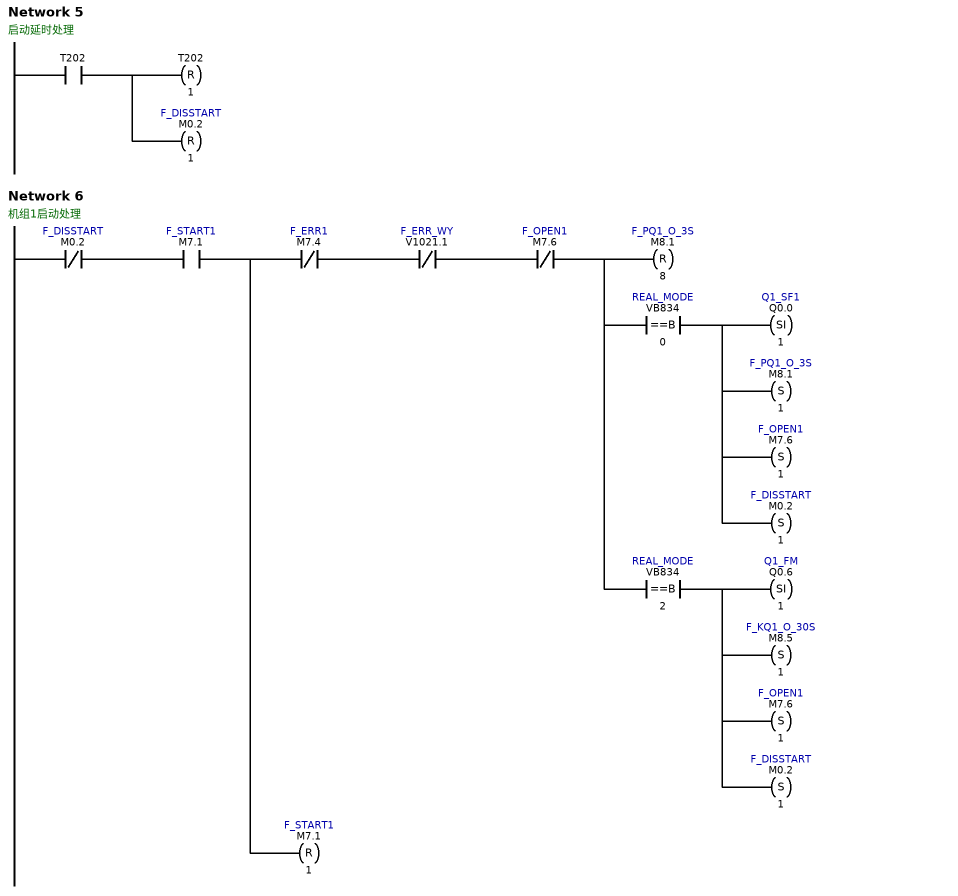
[picture p48: SBR7 networks 5-6]
Network 5
// 启动延时处理
LD     T202
R      T202, 1
R      F_DISSTART:M0.2, 1
Network 6
// 机组1启动处理
LDN    F_DISSTART:M0.2
A      F_START1:M7.1
LPS
AN     F_ERR1:M7.4
AN     F_ERR_WY:V1021.1
AN     F_OPEN1:M7.6
LPS
R      F_PQ1_O_3S:M8.1, 8
AB=    REAL_MODE:VB834, 0
SI     Q1_SF1:Q0.0, 1
S      F_PQ1_O_3S:M8.1, 1
S      F_OPEN1:M7.6, 1
S      F_DISSTART:M0.2, 1
LPP
AB=    REAL_MODE:VB834, 2
SI     Q1_FM:Q0.6, 1
S      F_KQ1_O_30S:M8.5, 1
S      F_OPEN1:M7.6, 1
S      F_DISSTART:M0.2, 1
LPP
R      F_START1:M7.1, 1
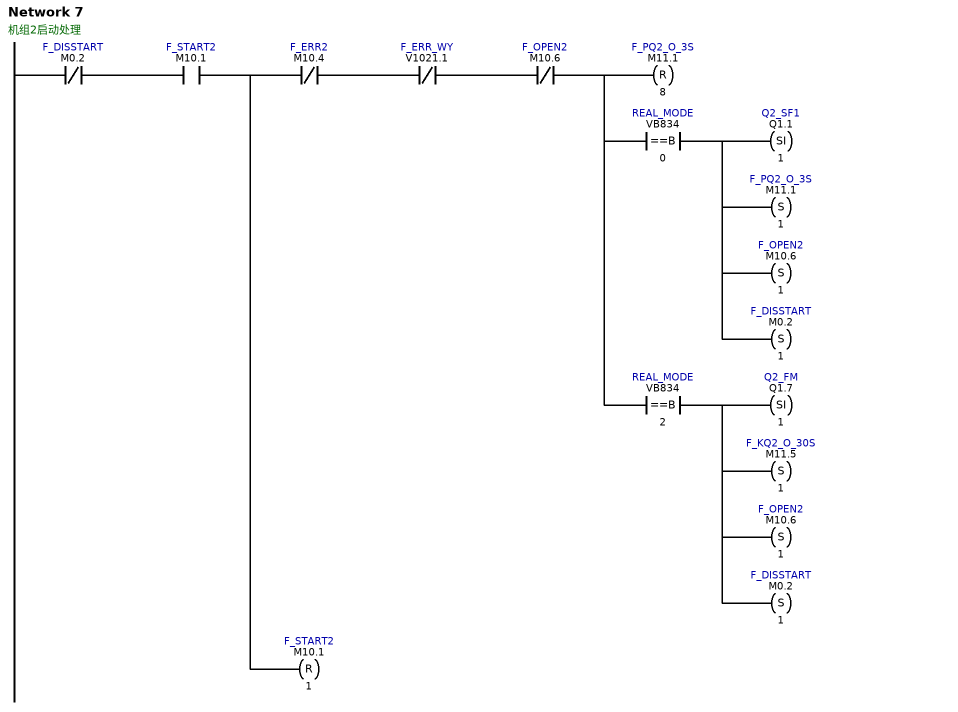
Network 7
// 机组2启动处理
LDN    F_DISSTART:M0.2
A      F_START2:M10.1
LPS
AN     F_ERR2:M10.4
AN     F_ERR_WY:V1021.1
AN     F_OPEN2:M10.6
LPS
R      F_PQ2_O_3S:M11.1, 8
AB=    REAL_MODE:VB834, 0
SI     Q2_SF1:Q1.1, 1
S      F_PQ2_O_3S:M11.1, 1
S      F_OPEN2:M10.6, 1
S      F_DISSTART:M0.2, 1
LPP
AB=    REAL_MODE:VB834, 2
SI     Q2_FM:Q1.7, 1
S      F_KQ2_O_30S:M11.5, 1
S      F_OPEN2:M10.6, 1
S      F_DISSTART:M0.2, 1
LPP
R      F_START2:M10.1, 1
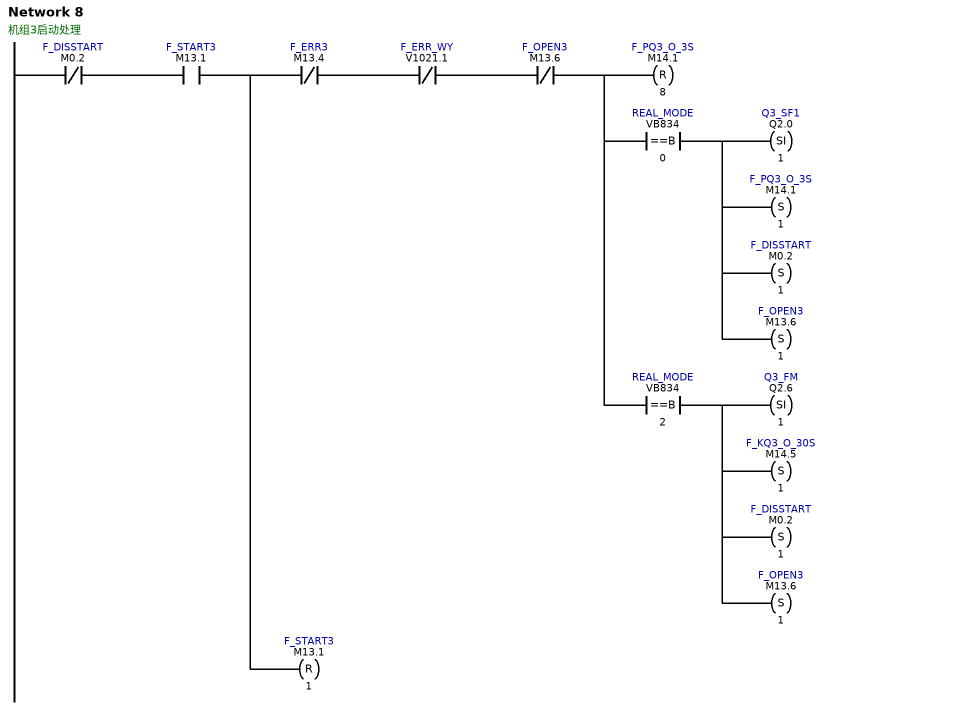
Network 8
// 机组3启动处理
LDN    F_DISSTART:M0.2
A      F_START3:M13.1
LPS
AN     F_ERR3:M13.4
AN     F_ERR_WY:V1021.1
AN     F_OPEN3:M13.6
LPS
R      F_PQ3_O_3S:M14.1, 8
AB=    REAL_MODE:VB834, 0
SI     Q3_SF1:Q2.0, 1
S      F_PQ3_O_3S:M14.1, 1
S      F_DISSTART:M0.2, 1
S      F_OPEN3:M13.6, 1
LPP
AB=    REAL_MODE:VB834, 2
SI     Q3_FM:Q2.6, 1
S      F_KQ3_O_30S:M14.5, 1
S      F_DISSTART:M0.2, 1
S      F_OPEN3:M13.6, 1
LPP
R      F_START3:M13.1, 1
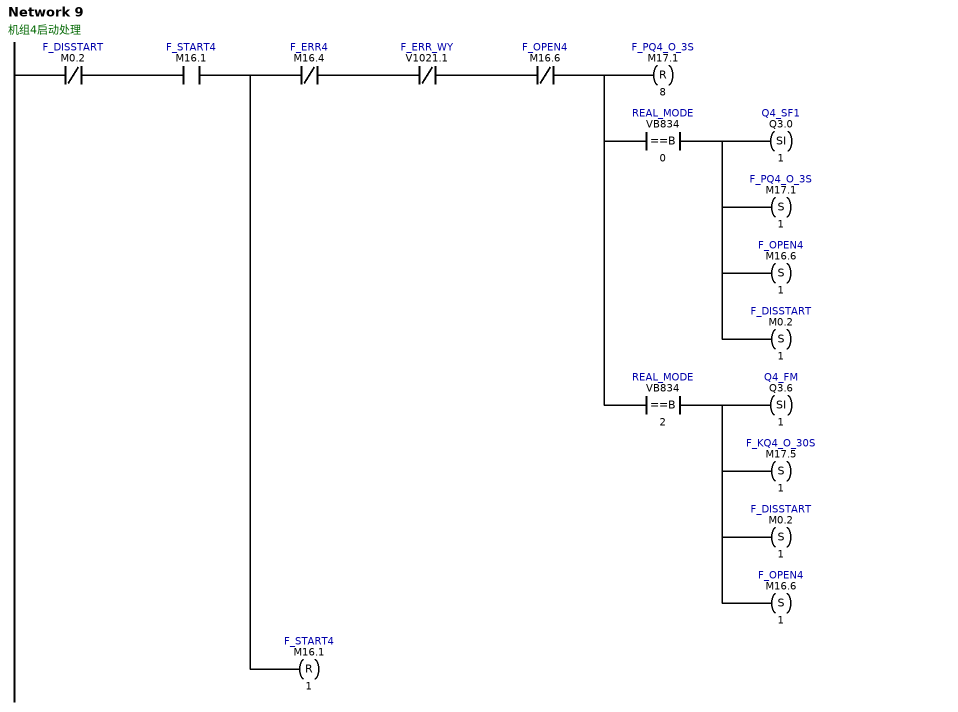
Network 9
// 机组4启动处理
LDN    F_DISSTART:M0.2
A      F_START4:M16.1
LPS
AN     F_ERR4:M16.4
AN     F_ERR_WY:V1021.1
AN     F_OPEN4:M16.6
LPS
R      F_PQ4_O_3S:M17.1, 8
AB=    REAL_MODE:VB834, 0
SI     Q4_SF1:Q3.0, 1
S      F_PQ4_O_3S:M17.1, 1
S      F_OPEN4:M16.6, 1
S      F_DISSTART:M0.2, 1
LPP
AB=    REAL_MODE:VB834, 2
SI     Q4_FM:Q3.6, 1
S      F_KQ4_O_30S:M17.5, 1
S      F_DISSTART:M0.2, 1
S      F_OPEN4:M16.6, 1
LPP
R      F_START4:M16.1, 1
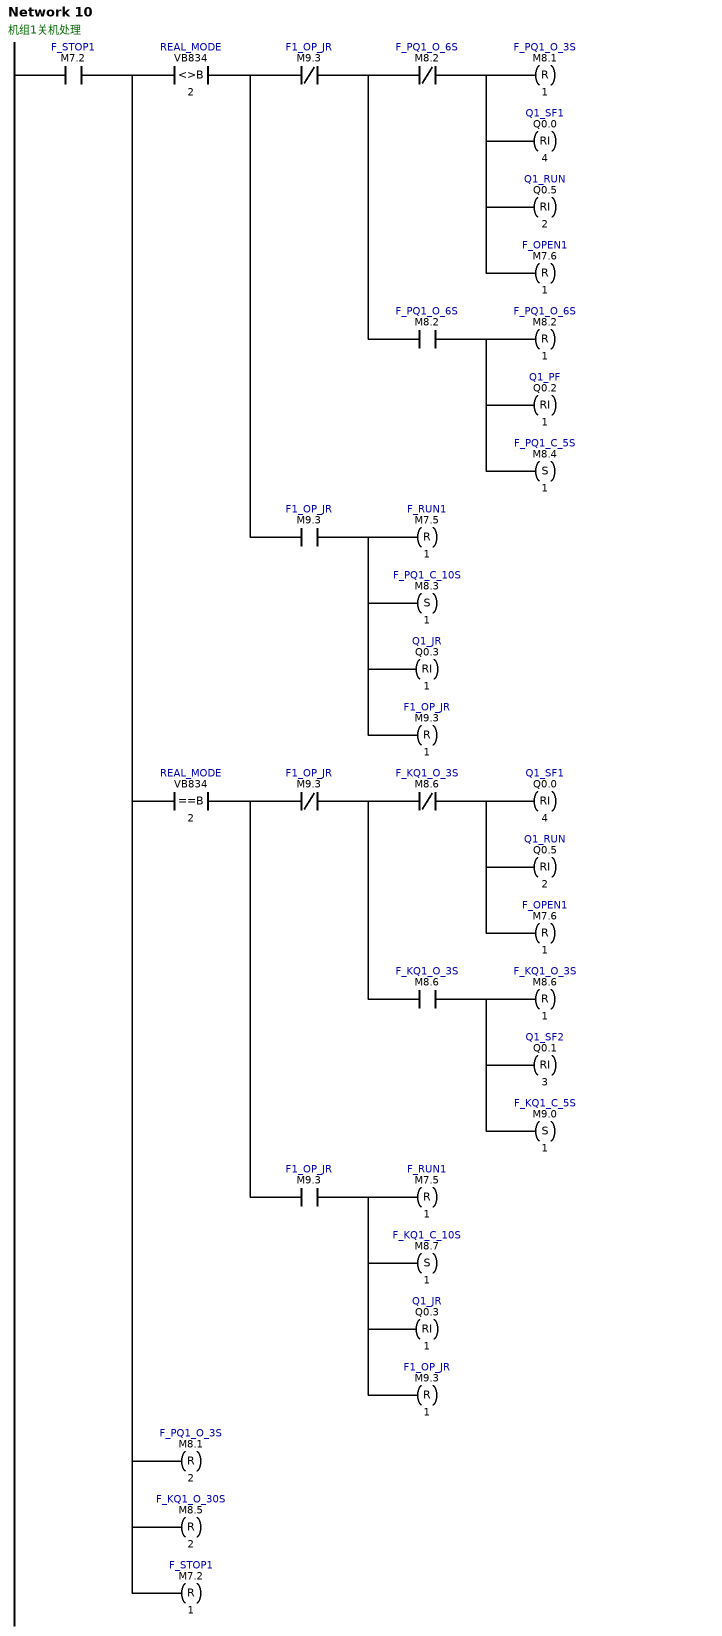
Network 10
// 机组1关机处理
LD     F_STOP1:M7.2
LPS
AB<>   REAL_MODE:VB834, 2
LPS
AN     F1_OP_JR:M9.3
LPS
AN     F_PQ1_O_6S:M8.2
R      F_PQ1_O_3S:M8.1, 1
RI     Q1_SF1:Q0.0, 4
RI     Q1_RUN:Q0.5, 2
R      F_OPEN1:M7.6, 1
LPP
A      F_PQ1_O_6S:M8.2
R      F_PQ1_O_6S:M8.2, 1
RI     Q1_PF:Q0.2, 1
S      F_PQ1_C_5S:M8.4, 1
LPP
A      F1_OP_JR:M9.3
R      F_RUN1:M7.5, 1
S      F_PQ1_C_10S:M8.3, 1
RI     Q1_JR:Q0.3, 1
R      F1_OP_JR:M9.3, 1
LRD
AB=    REAL_MODE:VB834, 2
LPS
AN     F1_OP_JR:M9.3
LPS
AN     F_KQ1_O_3S:M8.6
RI     Q1_SF1:Q0.0, 4
RI     Q1_RUN:Q0.5, 2
R      F_OPEN1:M7.6, 1
LPP
A      F_KQ1_O_3S:M8.6
R      F_KQ1_O_3S:M8.6, 1
RI     Q1_SF2:Q0.1, 3
S      F_KQ1_C_5S:M9.0, 1
LPP
A      F1_OP_JR:M9.3
R      F_RUN1:M7.5, 1
S      F_KQ1_C_10S:M8.7, 1
RI     Q1_JR:Q0.3, 1
R      F1_OP_JR:M9.3, 1
LPP
R      F_PQ1_O_3S:M8.1, 2
R      F_KQ1_O_30S:M8.5, 2
R      F_STOP1:M7.2, 1
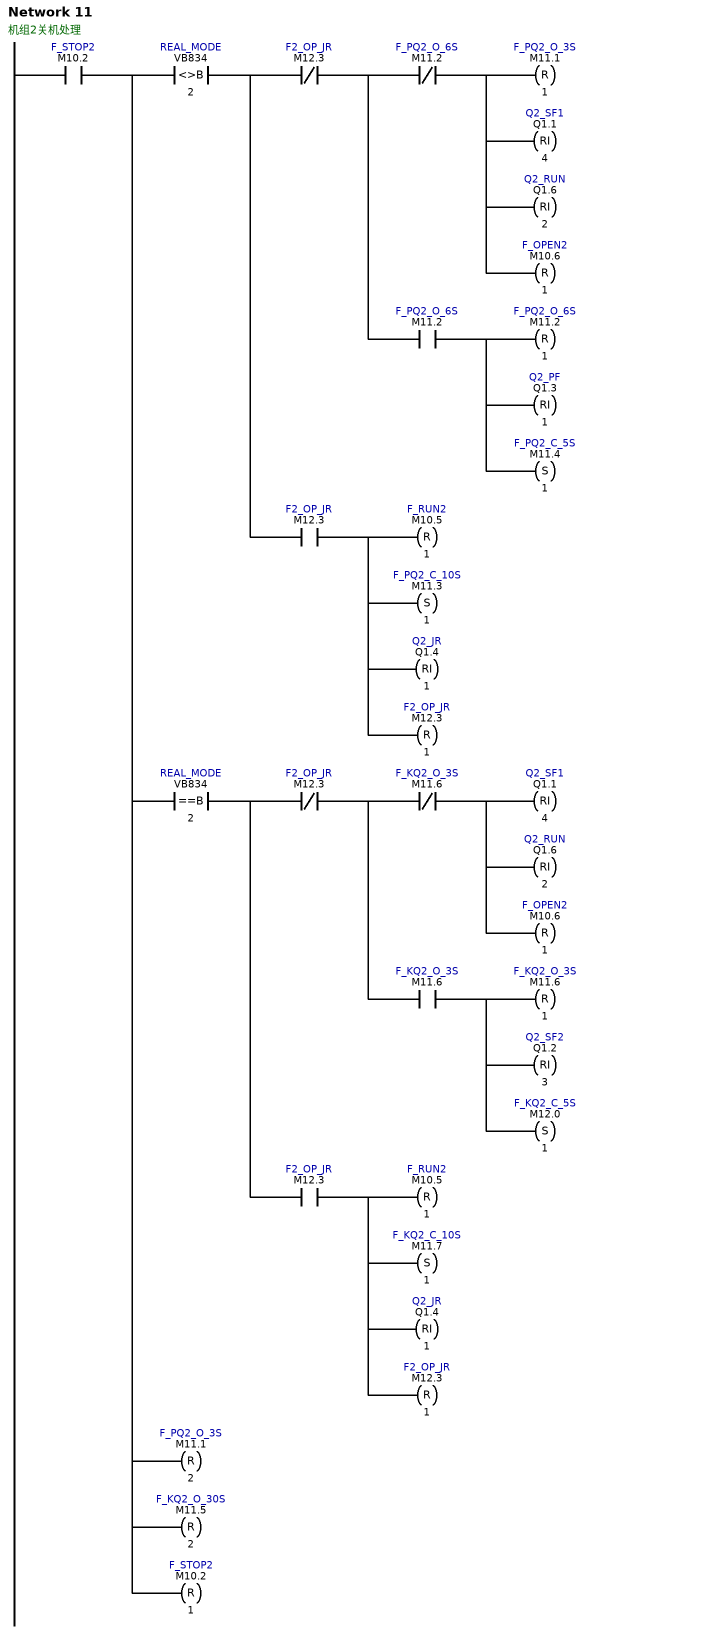
Network 11
// 机组2关机处理
LD     F_STOP2:M10.2
LPS
AB<>   REAL_MODE:VB834, 2
LPS
AN     F2_OP_JR:M12.3
LPS
AN     F_PQ2_O_6S:M11.2
R      F_PQ2_O_3S:M11.1, 1
RI     Q2_SF1:Q1.1, 4
RI     Q2_RUN:Q1.6, 2
R      F_OPEN2:M10.6, 1
LPP
A      F_PQ2_O_6S:M11.2
R      F_PQ2_O_6S:M11.2, 1
RI     Q2_PF:Q1.3, 1
S      F_PQ2_C_5S:M11.4, 1
LPP
A      F2_OP_JR:M12.3
R      F_RUN2:M10.5, 1
S      F_PQ2_C_10S:M11.3, 1
RI     Q2_JR:Q1.4, 1
R      F2_OP_JR:M12.3, 1
LRD
AB=    REAL_MODE:VB834, 2
LPS
AN     F2_OP_JR:M12.3
LPS
AN     F_KQ2_O_3S:M11.6
RI     Q2_SF1:Q1.1, 4
RI     Q2_RUN:Q1.6, 2
R      F_OPEN2:M10.6, 1
LPP
A      F_KQ2_O_3S:M11.6
R      F_KQ2_O_3S:M11.6, 1
RI     Q2_SF2:Q1.2, 3
S      F_KQ2_C_5S:M12.0, 1
LPP
A      F2_OP_JR:M12.3
R      F_RUN2:M10.5, 1
S      F_KQ2_C_10S:M11.7, 1
RI     Q2_JR:Q1.4, 1
R      F2_OP_JR:M12.3, 1
LPP
R      F_PQ2_O_3S:M11.1, 2
R      F_KQ2_O_30S:M11.5, 2
R      F_STOP2:M10.2, 1
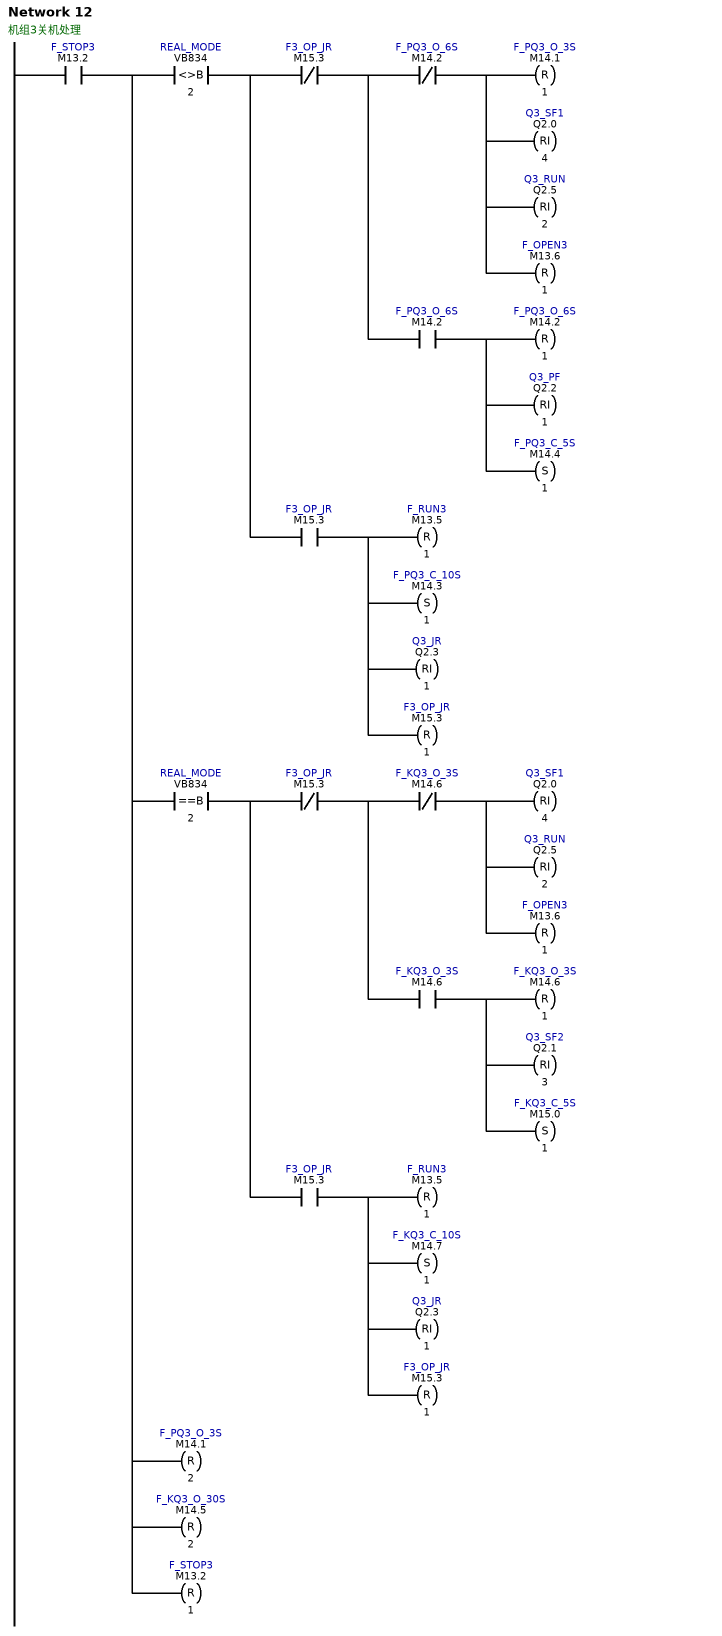
Network 12
// 机组3关机处理
LD     F_STOP3:M13.2
LPS
AB<>   REAL_MODE:VB834, 2
LPS
AN     F3_OP_JR:M15.3
LPS
AN     F_PQ3_O_6S:M14.2
R      F_PQ3_O_3S:M14.1, 1
RI     Q3_SF1:Q2.0, 4
RI     Q3_RUN:Q2.5, 2
R      F_OPEN3:M13.6, 1
LPP
A      F_PQ3_O_6S:M14.2
R      F_PQ3_O_6S:M14.2, 1
RI     Q3_PF:Q2.2, 1
S      F_PQ3_C_5S:M14.4, 1
LPP
A      F3_OP_JR:M15.3
R      F_RUN3:M13.5, 1
S      F_PQ3_C_10S:M14.3, 1
RI     Q3_JR:Q2.3, 1
R      F3_OP_JR:M15.3, 1
LRD
AB=    REAL_MODE:VB834, 2
LPS
AN     F3_OP_JR:M15.3
LPS
AN     F_KQ3_O_3S:M14.6
RI     Q3_SF1:Q2.0, 4
RI     Q3_RUN:Q2.5, 2
R      F_OPEN3:M13.6, 1
LPP
A      F_KQ3_O_3S:M14.6
R      F_KQ3_O_3S:M14.6, 1
RI     Q3_SF2:Q2.1, 3
S      F_KQ3_C_5S:M15.0, 1
LPP
A      F3_OP_JR:M15.3
R      F_RUN3:M13.5, 1
S      F_KQ3_C_10S:M14.7, 1
RI     Q3_JR:Q2.3, 1
R      F3_OP_JR:M15.3, 1
LPP
R      F_PQ3_O_3S:M14.1, 2
R      F_KQ3_O_30S:M14.5, 2
R      F_STOP3:M13.2, 1
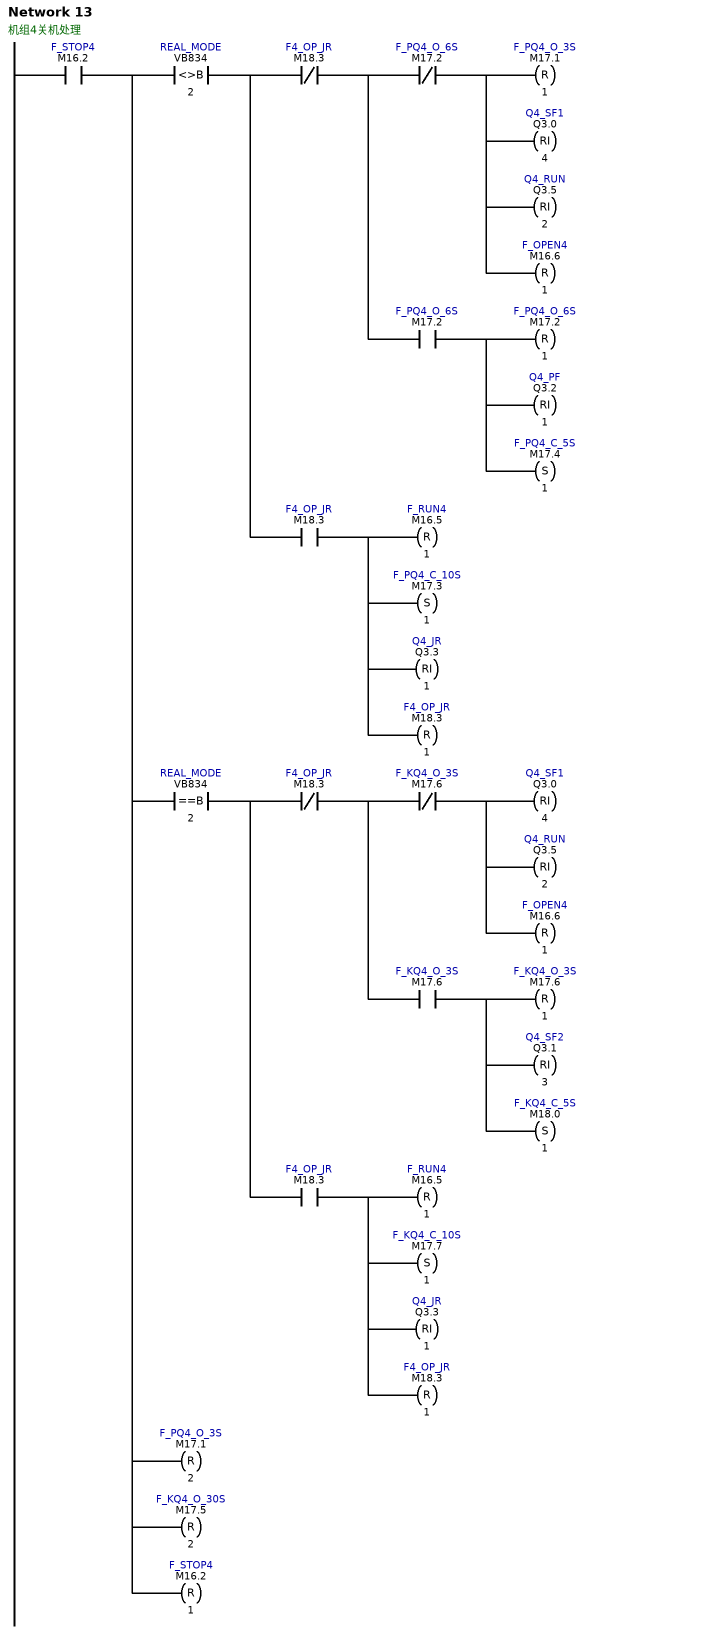
Network 13
// 机组4关机处理
LD     F_STOP4:M16.2
LPS
AB<>   REAL_MODE:VB834, 2
LPS
AN     F4_OP_JR:M18.3
LPS
AN     F_PQ4_O_6S:M17.2
R      F_PQ4_O_3S:M17.1, 1
RI     Q4_SF1:Q3.0, 4
RI     Q4_RUN:Q3.5, 2
R      F_OPEN4:M16.6, 1
LPP
A      F_PQ4_O_6S:M17.2
R      F_PQ4_O_6S:M17.2, 1
RI     Q4_PF:Q3.2, 1
S      F_PQ4_C_5S:M17.4, 1
LPP
A      F4_OP_JR:M18.3
R      F_RUN4:M16.5, 1
S      F_PQ4_C_10S:M17.3, 1
RI     Q4_JR:Q3.3, 1
R      F4_OP_JR:M18.3, 1
LRD
AB=    REAL_MODE:VB834, 2
LPS
AN     F4_OP_JR:M18.3
LPS
AN     F_KQ4_O_3S:M17.6
RI     Q4_SF1:Q3.0, 4
RI     Q4_RUN:Q3.5, 2
R      F_OPEN4:M16.6, 1
LPP
A      F_KQ4_O_3S:M17.6
R      F_KQ4_O_3S:M17.6, 1
RI     Q4_SF2:Q3.1, 3
S      F_KQ4_C_5S:M18.0, 1
LPP
A      F4_OP_JR:M18.3
R      F_RUN4:M16.5, 1
S      F_KQ4_C_10S:M17.7, 1
RI     Q4_JR:Q3.3, 1
R      F4_OP_JR:M18.3, 1
LPP
R      F_PQ4_O_3S:M17.1, 2
R      F_KQ4_O_30S:M17.5, 2
R      F_STOP4:M16.2, 1
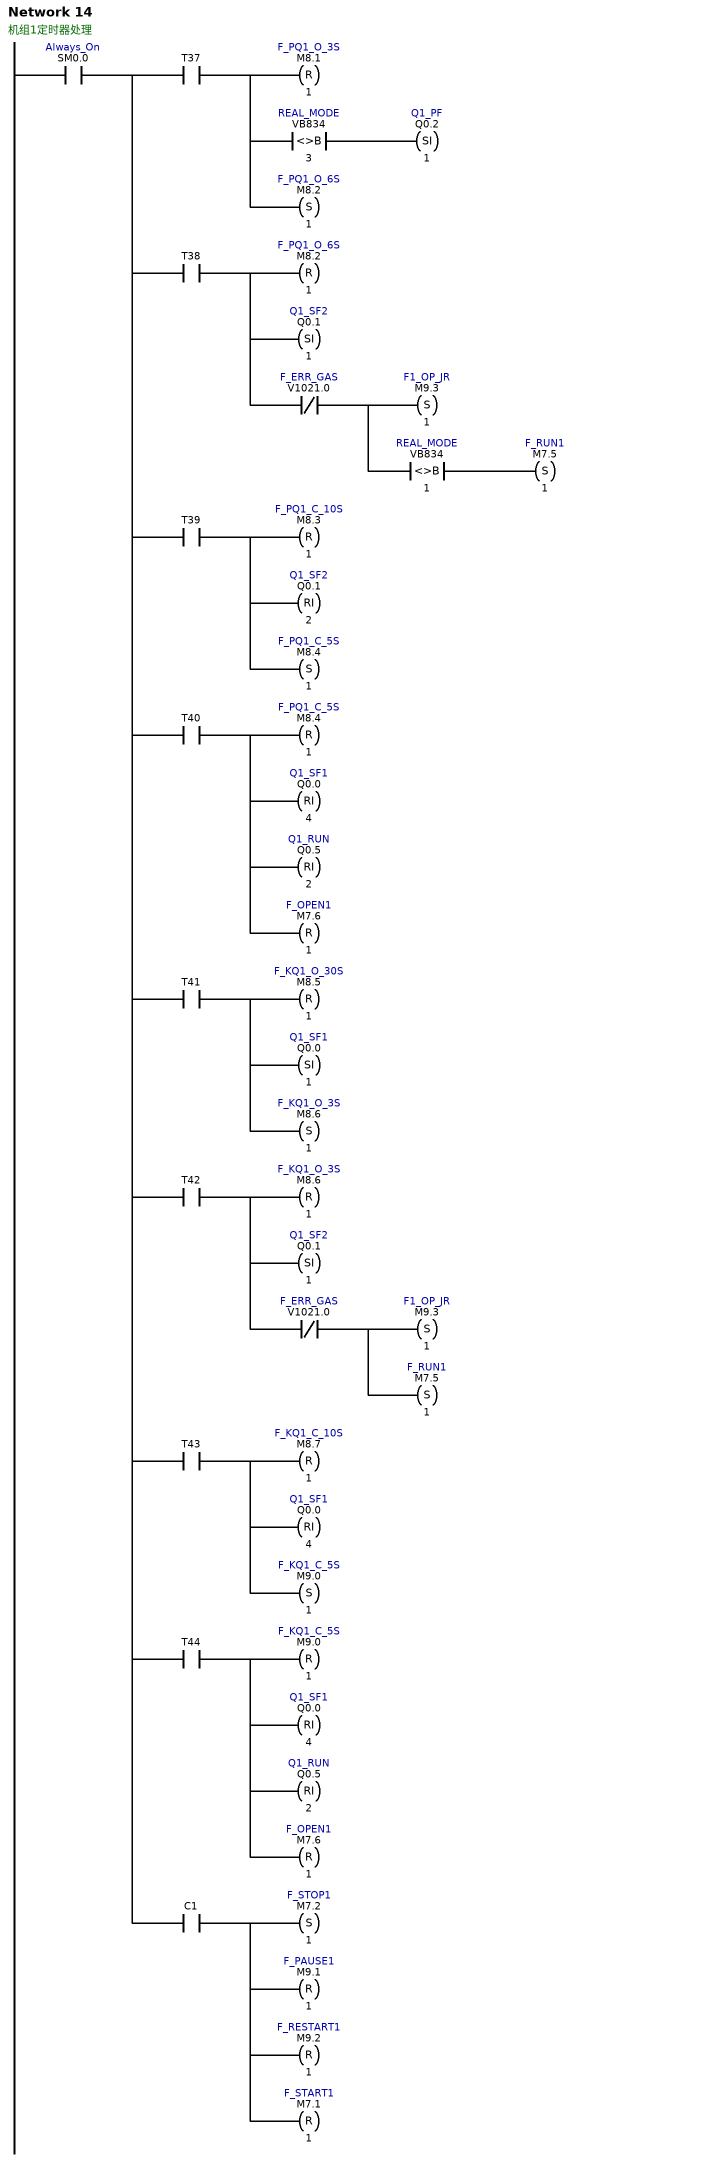
Network 14
// 机组1定时器处理
LD     Always_On:SM0.0
LPS
A      T37
LPS
R      F_PQ1_O_3S:M8.1, 1
AB<>   REAL_MODE:VB834, 3
SI     Q1_PF:Q0.2, 1
LPP
S      F_PQ1_O_6S:M8.2, 1
LRD
A      T38
R      F_PQ1_O_6S:M8.2, 1
SI     Q1_SF2:Q0.1, 1
AN     F_ERR_GAS:V1021.0
S      F1_OP_JR:M9.3, 1
AB<>   REAL_MODE:VB834, 1
S      F_RUN1:M7.5, 1
LRD
LPS
A      T39
R      F_PQ1_C_10S:M8.3, 1
RI     Q1_SF2:Q0.1, 2
S      F_PQ1_C_5S:M8.4, 1
LRD
A      T40
R      F_PQ1_C_5S:M8.4, 1
RI     Q1_SF1:Q0.0, 4
RI     Q1_RUN:Q0.5, 2
R      F_OPEN1:M7.6, 1
LPP
A      T41
R      F_KQ1_O_30S:M8.5, 1
SI     Q1_SF1:Q0.0, 1
S      F_KQ1_O_3S:M8.6, 1
LRD
A      T42
R      F_KQ1_O_3S:M8.6, 1
SI     Q1_SF2:Q0.1, 1
AN     F_ERR_GAS:V1021.0
S      F1_OP_JR:M9.3, 1
S      F_RUN1:M7.5, 1
LPP
LPS
A      T43
R      F_KQ1_C_10S:M8.7, 1
RI     Q1_SF1:Q0.0, 4
S      F_KQ1_C_5S:M9.0, 1
LRD
A      T44
R      F_KQ1_C_5S:M9.0, 1
RI     Q1_SF1:Q0.0, 4
RI     Q1_RUN:Q0.5, 2
R      F_OPEN1:M7.6, 1
LPP
A      C1
S      F_STOP1:M7.2, 1
R      F_PAUSE1:M9.1, 1
R      F_RESTART1:M9.2, 1
R      F_START1:M7.1, 1
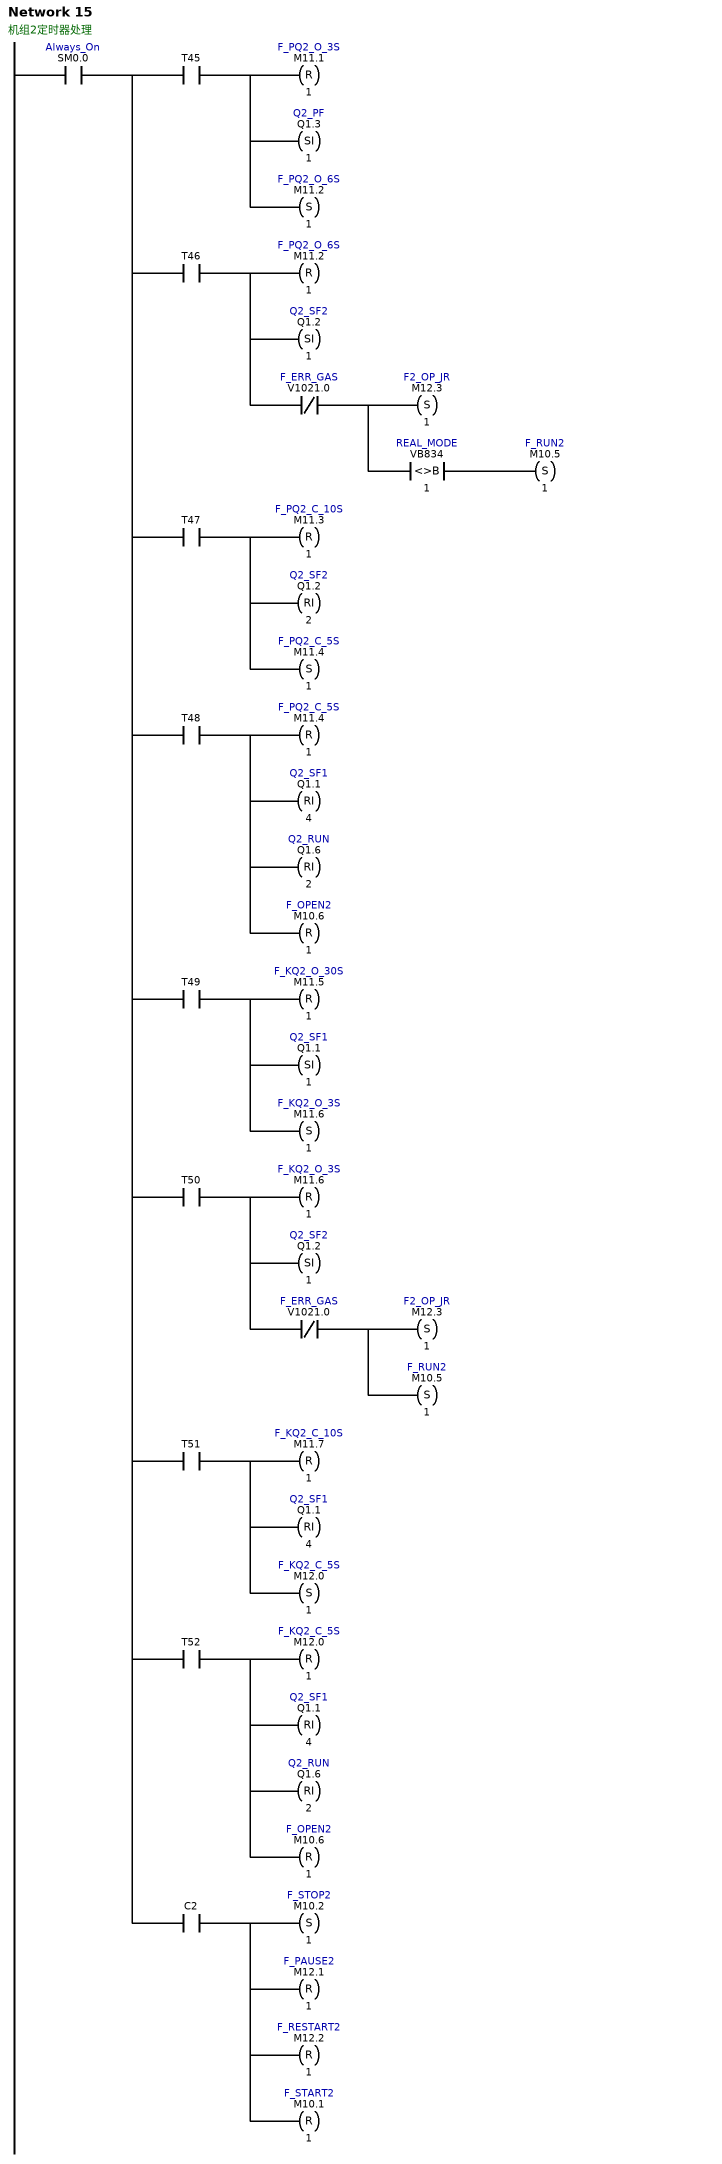
Network 15
// 机组2定时器处理
LD     Always_On:SM0.0
LPS
A      T45
R      F_PQ2_O_3S:M11.1, 1
SI     Q2_PF:Q1.3, 1
S      F_PQ2_O_6S:M11.2, 1
LRD
A      T46
R      F_PQ2_O_6S:M11.2, 1
SI     Q2_SF2:Q1.2, 1
AN     F_ERR_GAS:V1021.0
S      F2_OP_JR:M12.3, 1
AB<>   REAL_MODE:VB834, 1
S      F_RUN2:M10.5, 1
LRD
LPS
A      T47
R      F_PQ2_C_10S:M11.3, 1
RI     Q2_SF2:Q1.2, 2
S      F_PQ2_C_5S:M11.4, 1
LRD
A      T48
R      F_PQ2_C_5S:M11.4, 1
RI     Q2_SF1:Q1.1, 4
RI     Q2_RUN:Q1.6, 2
R      F_OPEN2:M10.6, 1
LPP
A      T49
R      F_KQ2_O_30S:M11.5, 1
SI     Q2_SF1:Q1.1, 1
S      F_KQ2_O_3S:M11.6, 1
LRD
A      T50
R      F_KQ2_O_3S:M11.6, 1
SI     Q2_SF2:Q1.2, 1
AN     F_ERR_GAS:V1021.0
S      F2_OP_JR:M12.3, 1
S      F_RUN2:M10.5, 1
LPP
LPS
A      T51
R      F_KQ2_C_10S:M11.7, 1
RI     Q2_SF1:Q1.1, 4
S      F_KQ2_C_5S:M12.0, 1
LRD
A      T52
R      F_KQ2_C_5S:M12.0, 1
RI     Q2_SF1:Q1.1, 4
RI     Q2_RUN:Q1.6, 2
R      F_OPEN2:M10.6, 1
LPP
A      C2
S      F_STOP2:M10.2, 1
R      F_PAUSE2:M12.1, 1
R      F_RESTART2:M12.2, 1
R      F_START2:M10.1, 1
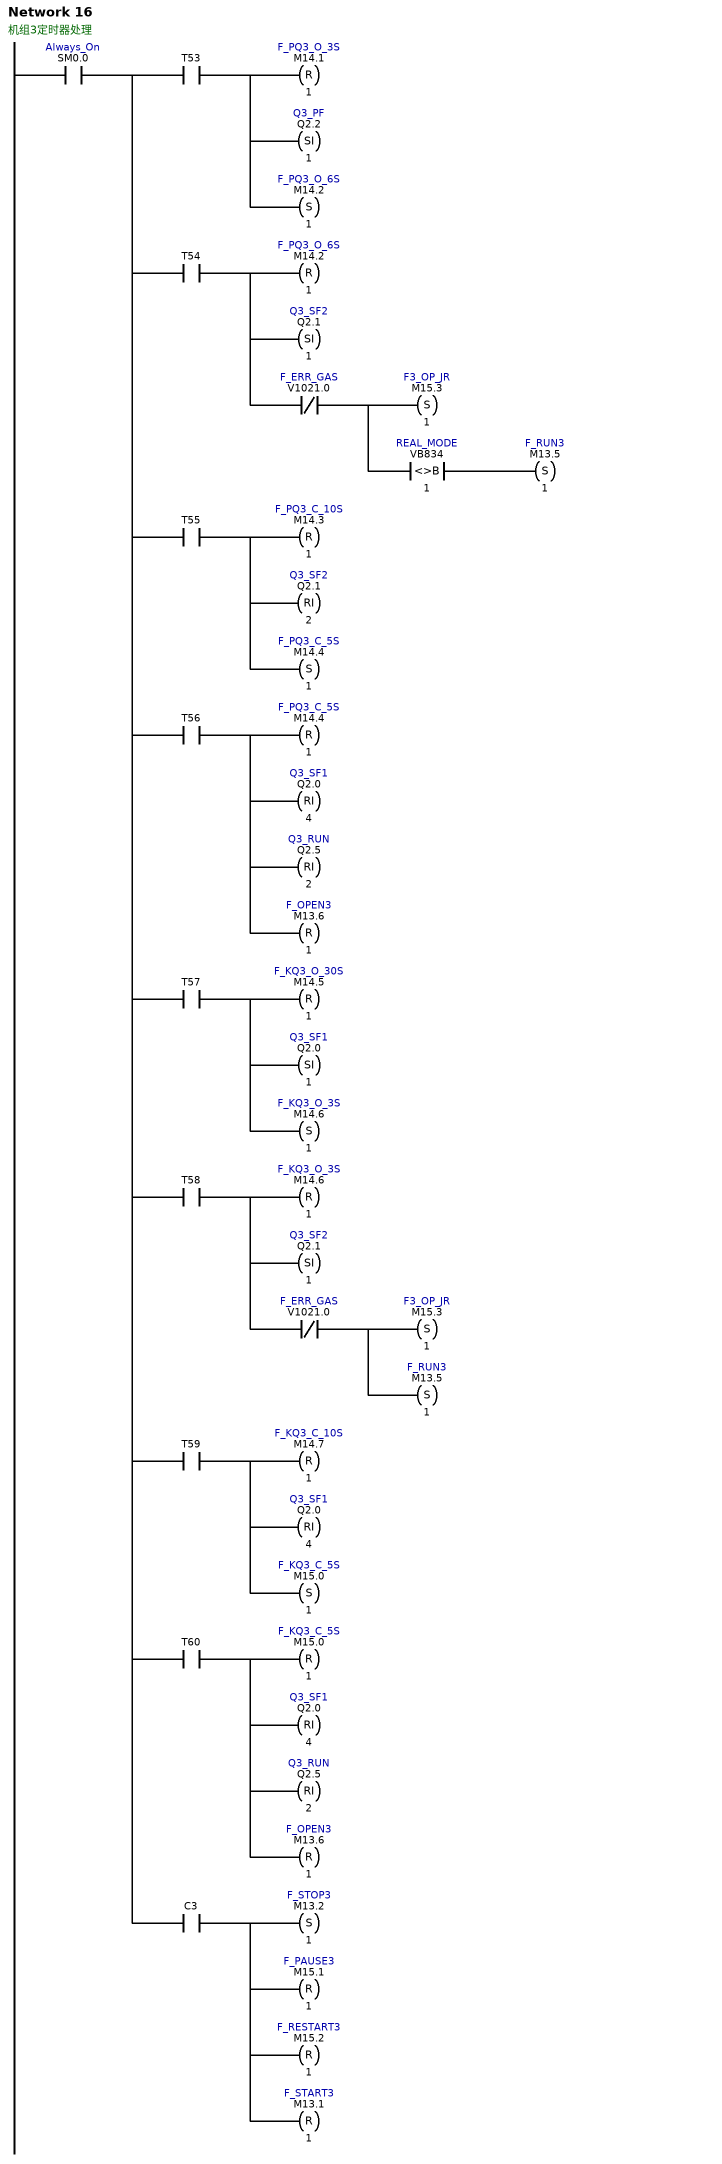
Network 16
// 机组3定时器处理
LD     Always_On:SM0.0
LPS
A      T53
R      F_PQ3_O_3S:M14.1, 1
SI     Q3_PF:Q2.2, 1
S      F_PQ3_O_6S:M14.2, 1
LRD
A      T54
R      F_PQ3_O_6S:M14.2, 1
SI     Q3_SF2:Q2.1, 1
AN     F_ERR_GAS:V1021.0
S      F3_OP_JR:M15.3, 1
AB<>   REAL_MODE:VB834, 1
S      F_RUN3:M13.5, 1
LRD
LPS
A      T55
R      F_PQ3_C_10S:M14.3, 1
RI     Q3_SF2:Q2.1, 2
S      F_PQ3_C_5S:M14.4, 1
LRD
A      T56
R      F_PQ3_C_5S:M14.4, 1
RI     Q3_SF1:Q2.0, 4
RI     Q3_RUN:Q2.5, 2
R      F_OPEN3:M13.6, 1
LPP
A      T57
R      F_KQ3_O_30S:M14.5, 1
SI     Q3_SF1:Q2.0, 1
S      F_KQ3_O_3S:M14.6, 1
LRD
A      T58
R      F_KQ3_O_3S:M14.6, 1
SI     Q3_SF2:Q2.1, 1
AN     F_ERR_GAS:V1021.0
S      F3_OP_JR:M15.3, 1
S      F_RUN3:M13.5, 1
LPP
LPS
A      T59
R      F_KQ3_C_10S:M14.7, 1
RI     Q3_SF1:Q2.0, 4
S      F_KQ3_C_5S:M15.0, 1
LRD
A      T60
R      F_KQ3_C_5S:M15.0, 1
RI     Q3_SF1:Q2.0, 4
RI     Q3_RUN:Q2.5, 2
R      F_OPEN3:M13.6, 1
LPP
A      C3
S      F_STOP3:M13.2, 1
R      F_PAUSE3:M15.1, 1
R      F_RESTART3:M15.2, 1
R      F_START3:M13.1, 1
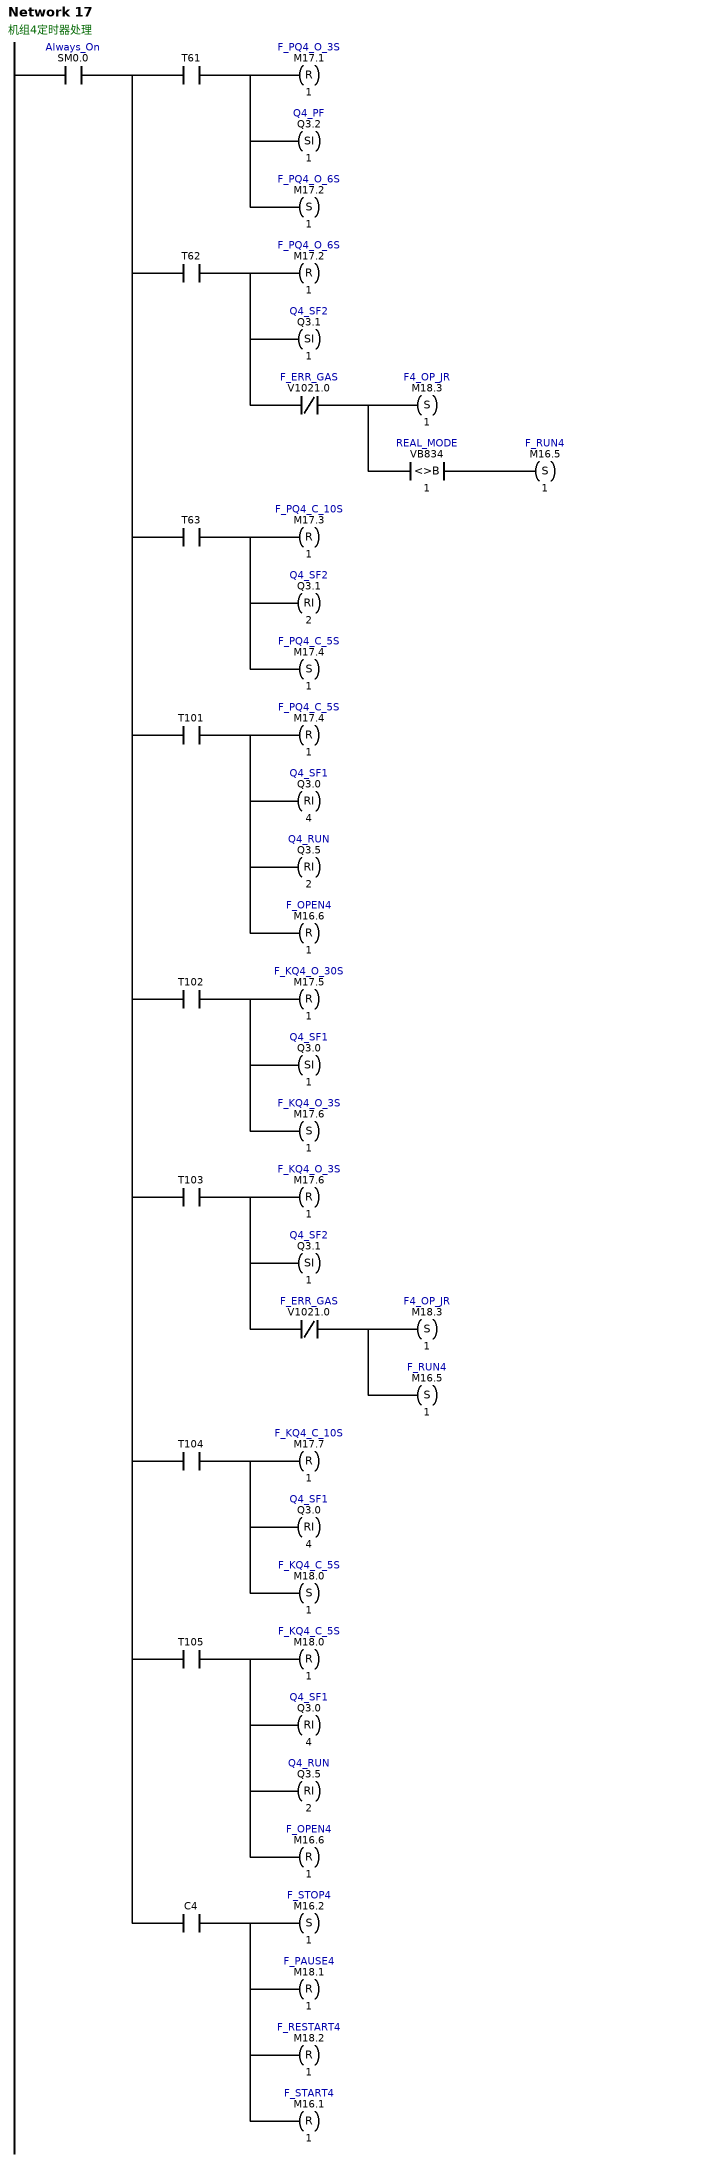
Network 17
// 机组4定时器处理
LD     Always_On:SM0.0
LPS
A      T61
R      F_PQ4_O_3S:M17.1, 1
SI     Q4_PF:Q3.2, 1
S      F_PQ4_O_6S:M17.2, 1
LRD
A      T62
R      F_PQ4_O_6S:M17.2, 1
SI     Q4_SF2:Q3.1, 1
AN     F_ERR_GAS:V1021.0
S      F4_OP_JR:M18.3, 1
AB<>   REAL_MODE:VB834, 1
S      F_RUN4:M16.5, 1
LRD
LPS
A      T63
R      F_PQ4_C_10S:M17.3, 1
RI     Q4_SF2:Q3.1, 2
S      F_PQ4_C_5S:M17.4, 1
LRD
A      T101
R      F_PQ4_C_5S:M17.4, 1
RI     Q4_SF1:Q3.0, 4
RI     Q4_RUN:Q3.5, 2
R      F_OPEN4:M16.6, 1
LPP
A      T102
R      F_KQ4_O_30S:M17.5, 1
SI     Q4_SF1:Q3.0, 1
S      F_KQ4_O_3S:M17.6, 1
LRD
A      T103
R      F_KQ4_O_3S:M17.6, 1
SI     Q4_SF2:Q3.1, 1
AN     F_ERR_GAS:V1021.0
S      F4_OP_JR:M18.3, 1
S      F_RUN4:M16.5, 1
LPP
LPS
A      T104
R      F_KQ4_C_10S:M17.7, 1
RI     Q4_SF1:Q3.0, 4
S      F_KQ4_C_5S:M18.0, 1
LRD
A      T105
R      F_KQ4_C_5S:M18.0, 1
RI     Q4_SF1:Q3.0, 4
RI     Q4_RUN:Q3.5, 2
R      F_OPEN4:M16.6, 1
LPP
A      C4
S      F_STOP4:M16.2, 1
R      F_PAUSE4:M18.1, 1
R      F_RESTART4:M18.2, 1
R      F_START4:M16.1, 1
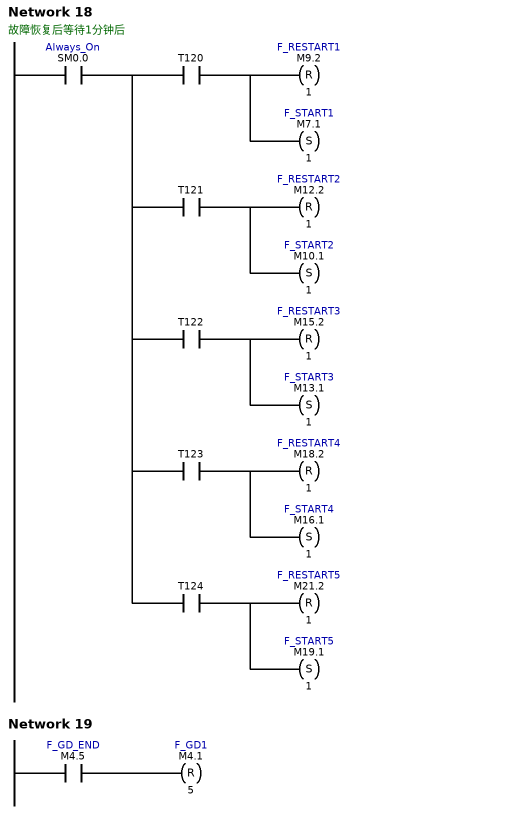
Network 18
// 故障恢复后等待1分钟后
LD     Always_On:SM0.0
LPS
A      T120
R      F_RESTART1:M9.2, 1
S      F_START1:M7.1, 1
LRD
A      T121
R      F_RESTART2:M12.2, 1
S      F_START2:M10.1, 1
LRD
A      T122
R      F_RESTART3:M15.2, 1
S      F_START3:M13.1, 1
LRD
A      T123
R      F_RESTART4:M18.2, 1
S      F_START4:M16.1, 1
LPP
A      T124
R      F_RESTART5:M21.2, 1
S      F_START5:M19.1, 1
Network 19
LD     F_GD_END:M4.5
R      F_GD1:M4.1, 5
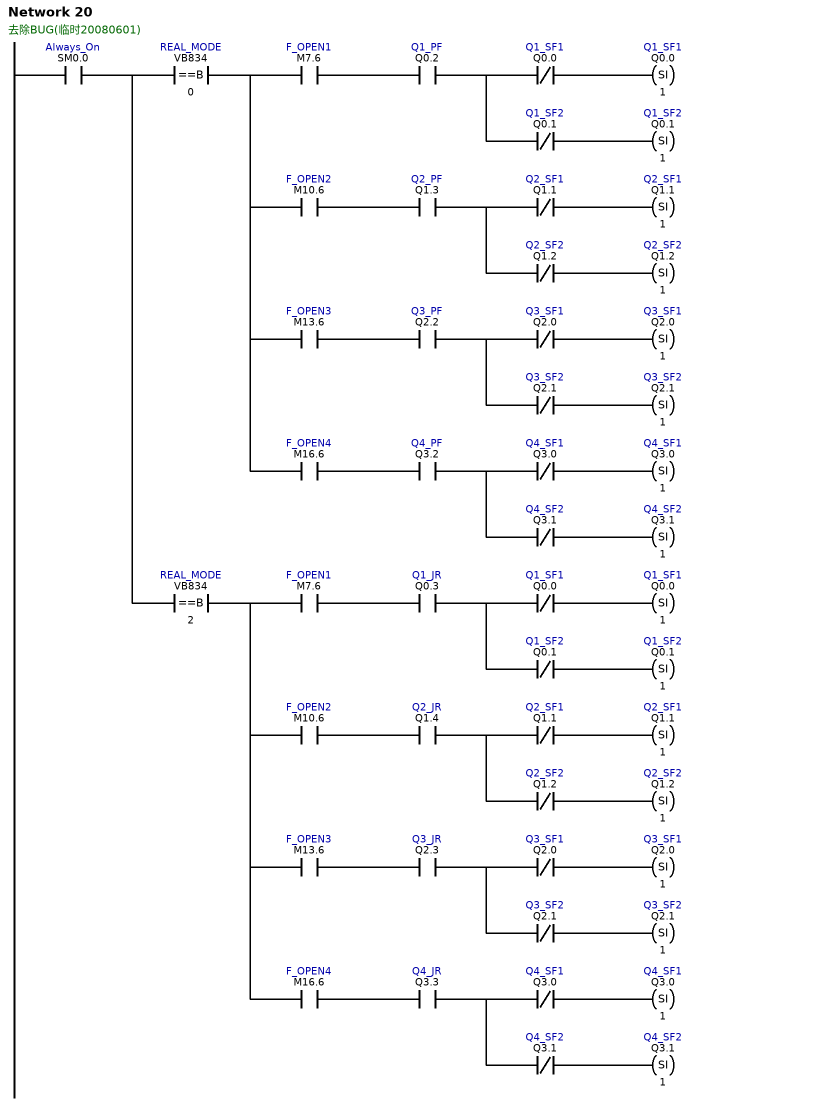
Network 20
// 去除BUG(临时20080601)
LD     Always_On:SM0.0
LPS
AB=    REAL_MODE:VB834, 0
LPS
A      F_OPEN1:M7.6
A      Q1_PF:Q0.2
LPS
AN     Q1_SF1:Q0.0
SI     Q1_SF1:Q0.0, 1
LPP
AN     Q1_SF2:Q0.1
SI     Q1_SF2:Q0.1, 1
LRD
A      F_OPEN2:M10.6
A      Q2_PF:Q1.3
LPS
AN     Q2_SF1:Q1.1
SI     Q2_SF1:Q1.1, 1
LPP
AN     Q2_SF2:Q1.2
SI     Q2_SF2:Q1.2, 1
LRD
A      F_OPEN3:M13.6
A      Q3_PF:Q2.2
LPS
AN     Q3_SF1:Q2.0
SI     Q3_SF1:Q2.0, 1
LPP
AN     Q3_SF2:Q2.1
SI     Q3_SF2:Q2.1, 1
LPP
A      F_OPEN4:M16.6
A      Q4_PF:Q3.2
LPS
AN     Q4_SF1:Q3.0
SI     Q4_SF1:Q3.0, 1
LPP
AN     Q4_SF2:Q3.1
SI     Q4_SF2:Q3.1, 1
LPP
AB=    REAL_MODE:VB834, 2
LPS
A      F_OPEN1:M7.6
A      Q1_JR:Q0.3
LPS
AN     Q1_SF1:Q0.0
SI     Q1_SF1:Q0.0, 1
LPP
AN     Q1_SF2:Q0.1
SI     Q1_SF2:Q0.1, 1
LRD
A      F_OPEN2:M10.6
A      Q2_JR:Q1.4
LPS
AN     Q2_SF1:Q1.1
SI     Q2_SF1:Q1.1, 1
LPP
AN     Q2_SF2:Q1.2
SI     Q2_SF2:Q1.2, 1
LRD
A      F_OPEN3:M13.6
A      Q3_JR:Q2.3
LPS
AN     Q3_SF1:Q2.0
SI     Q3_SF1:Q2.0, 1
LPP
AN     Q3_SF2:Q2.1
SI     Q3_SF2:Q2.1, 1
LPP
A      F_OPEN4:M16.6
A      Q4_JR:Q3.3
LPS
AN     Q4_SF1:Q3.0
SI     Q4_SF1:Q3.0, 1
LPP
AN     Q4_SF2:Q3.1
SI     Q4_SF2:Q3.1, 1
END_SUBROUTINE_BLOCK

SUBROUTINE_BLOCK 读EEPROM:SBR8
TITLE=
VAR
TEMP:DWORD;	// LD0 
END_VAR
BEGIN
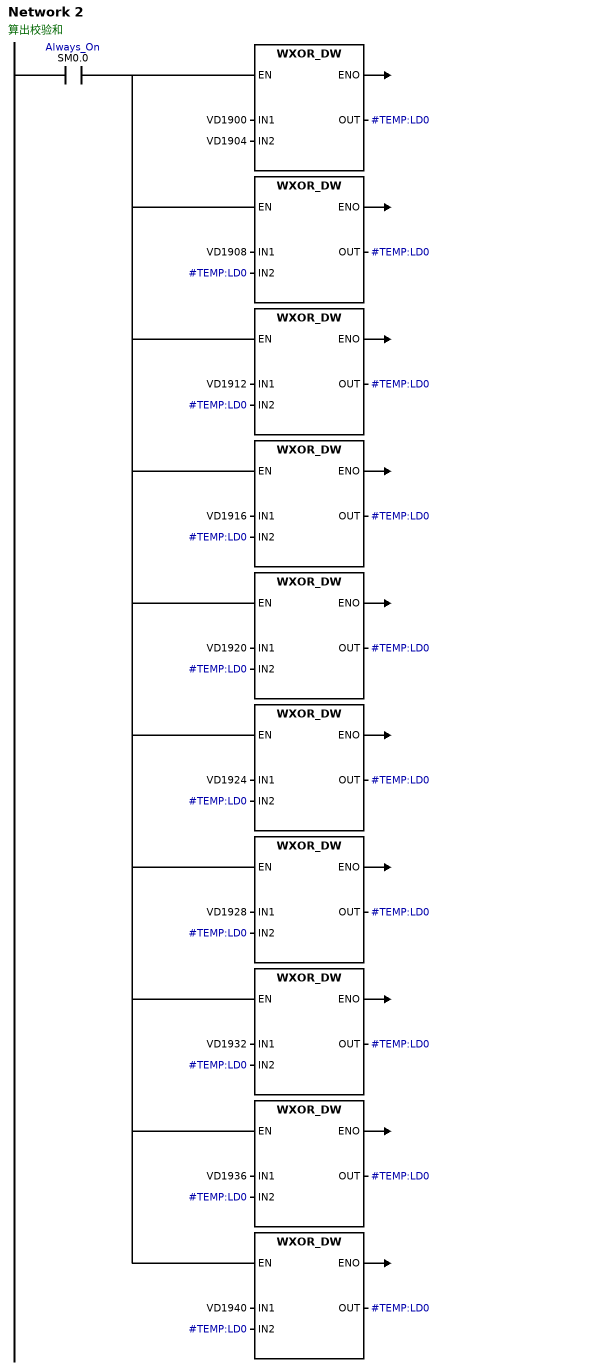
Network 2
// 算出校验和
LD     Always_On:SM0.0
MOVD   VD1900, #TEMP:LD0
XORD   VD1904, #TEMP:LD0
XORD   VD1908, #TEMP:LD0
XORD   VD1912, #TEMP:LD0
XORD   VD1916, #TEMP:LD0
XORD   VD1920, #TEMP:LD0
XORD   VD1924, #TEMP:LD0
XORD   VD1928, #TEMP:LD0
XORD   VD1932, #TEMP:LD0
XORD   VD1936, #TEMP:LD0
XORD   VD1940, #TEMP:LD0
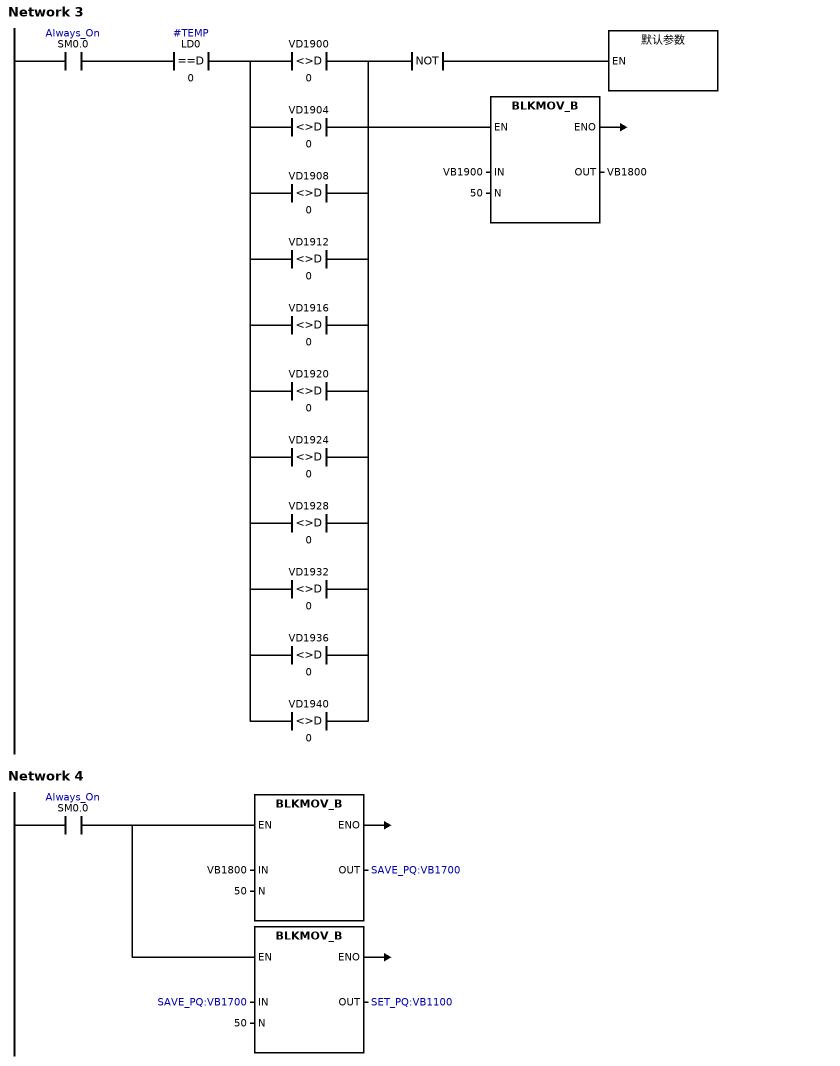
Network 3
LD     Always_On:SM0.0
AD=    #TEMP:LD0, 0
LDD<>  VD1900, 0
OD<>   VD1904, 0
OD<>   VD1908, 0
OD<>   VD1912, 0
OD<>   VD1916, 0
OD<>   VD1920, 0
OD<>   VD1924, 0
OD<>   VD1928, 0
OD<>   VD1932, 0
OD<>   VD1936, 0
OD<>   VD1940, 0
ALD
LPS
NOT
CALL   默认参数:SBR21
LPP
BMB    VB1900, VB1800, 50
Network 4
LD     Always_On:SM0.0
BMB    VB1800, SAVE_PQ:VB1700, 50
BMB    SAVE_PQ:VB1700, SET_PQ:VB1100, 50
END_SUBROUTINE_BLOCK

SUBROUTINE_BLOCK 定时器:SBR9
TITLE=
VAR
TEMP_W:WORD;	// LW0 
END_VAR
BEGIN
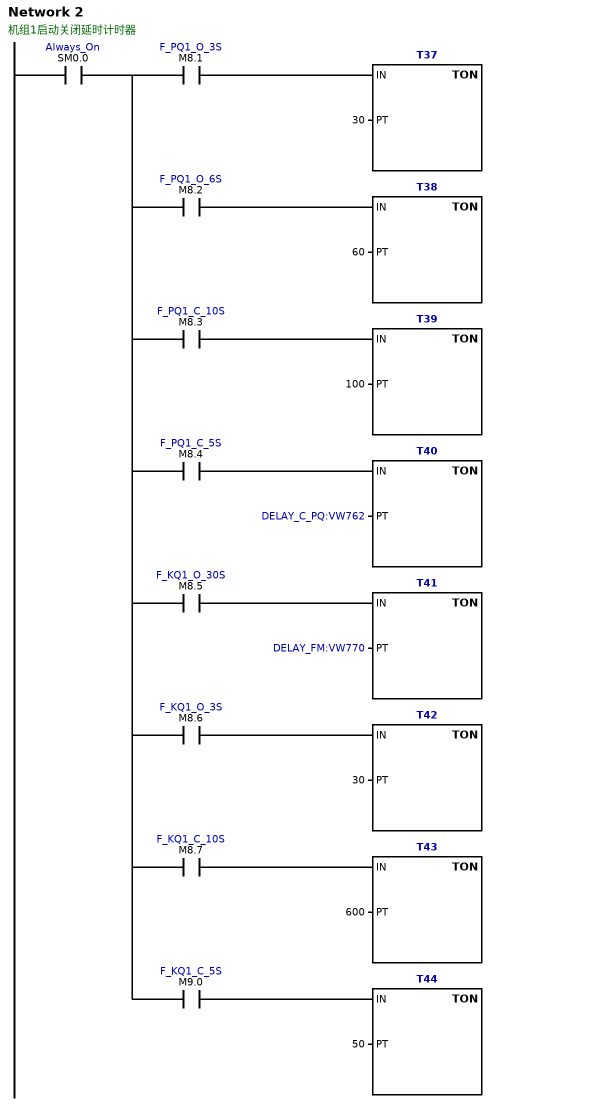
Network 2
// 机组1启动关闭延时计时器
LD     Always_On:SM0.0
LPS
A      F_PQ1_O_3S:M8.1
TON    T37, 30
LRD
A      F_PQ1_O_6S:M8.2
TON    T38, 60
LRD
A      F_PQ1_C_10S:M8.3
TON    T39, 100
LRD
A      F_PQ1_C_5S:M8.4
TON    T40, DELAY_C_PQ:VW762
LRD
A      F_KQ1_O_30S:M8.5
TON    T41, DELAY_FM:VW770
LRD
A      F_KQ1_O_3S:M8.6
TON    T42, 30
LRD
A      F_KQ1_C_10S:M8.7
TON    T43, 600
LPP
A      F_KQ1_C_5S:M9.0
TON    T44, 50
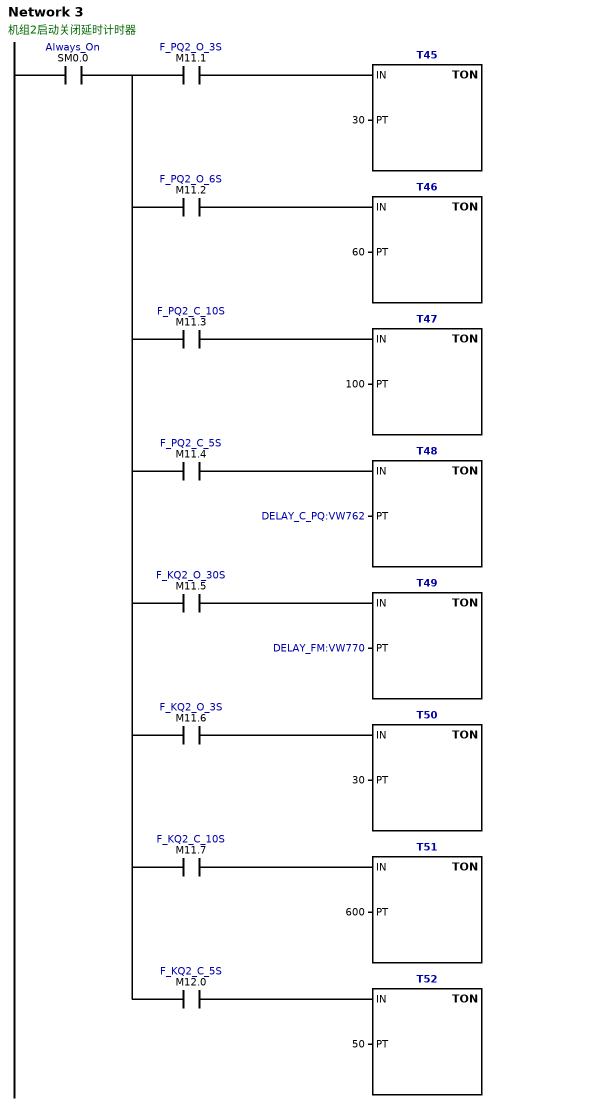
Network 3
// 机组2启动关闭延时计时器
LD     Always_On:SM0.0
LPS
A      F_PQ2_O_3S:M11.1
TON    T45, 30
LRD
A      F_PQ2_O_6S:M11.2
TON    T46, 60
LRD
A      F_PQ2_C_10S:M11.3
TON    T47, 100
LRD
A      F_PQ2_C_5S:M11.4
TON    T48, DELAY_C_PQ:VW762
LRD
A      F_KQ2_O_30S:M11.5
TON    T49, DELAY_FM:VW770
LRD
A      F_KQ2_O_3S:M11.6
TON    T50, 30
LRD
A      F_KQ2_C_10S:M11.7
TON    T51, 600
LPP
A      F_KQ2_C_5S:M12.0
TON    T52, 50
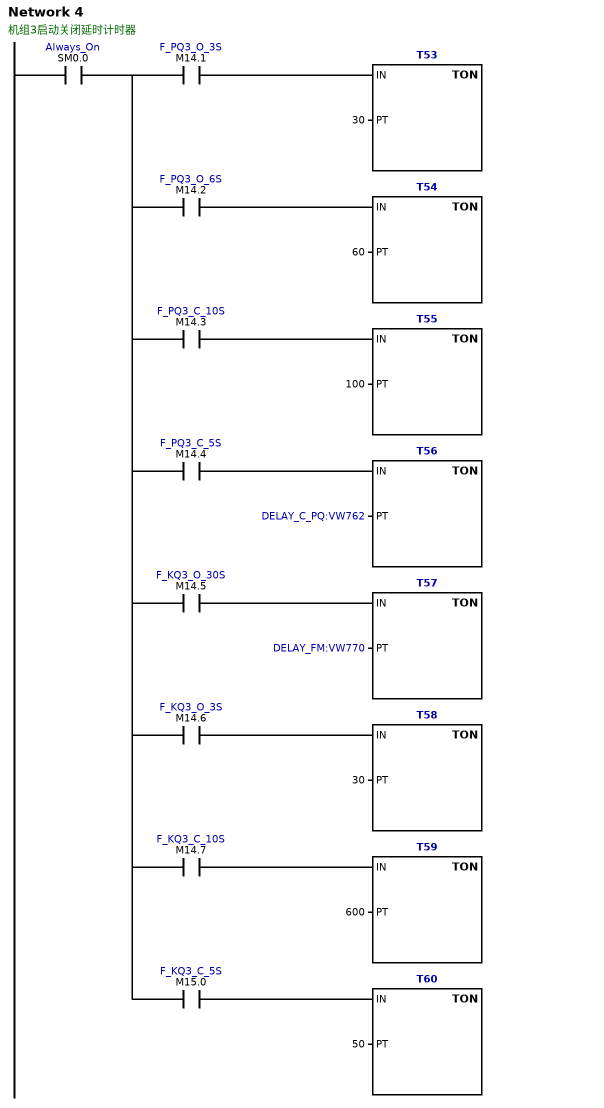
Network 4
// 机组3启动关闭延时计时器
LD     Always_On:SM0.0
LPS
A      F_PQ3_O_3S:M14.1
TON    T53, 30
LRD
A      F_PQ3_O_6S:M14.2
TON    T54, 60
LRD
A      F_PQ3_C_10S:M14.3
TON    T55, 100
LRD
A      F_PQ3_C_5S:M14.4
TON    T56, DELAY_C_PQ:VW762
LRD
A      F_KQ3_O_30S:M14.5
TON    T57, DELAY_FM:VW770
LRD
A      F_KQ3_O_3S:M14.6
TON    T58, 30
LRD
A      F_KQ3_C_10S:M14.7
TON    T59, 600
LPP
A      F_KQ3_C_5S:M15.0
TON    T60, 50
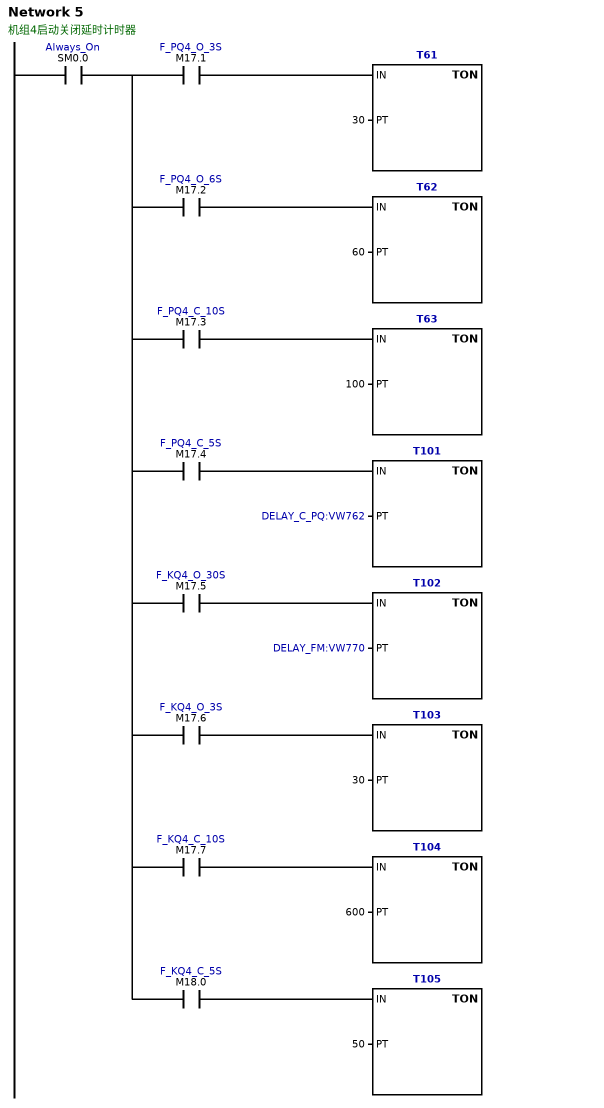
Network 5
// 机组4启动关闭延时计时器
LD     Always_On:SM0.0
LPS
A      F_PQ4_O_3S:M17.1
TON    T61, 30
LRD
A      F_PQ4_O_6S:M17.2
TON    T62, 60
LRD
A      F_PQ4_C_10S:M17.3
TON    T63, 100
LRD
A      F_PQ4_C_5S:M17.4
TON    T101, DELAY_C_PQ:VW762
LRD
A      F_KQ4_O_30S:M17.5
TON    T102, DELAY_FM:VW770
LRD
A      F_KQ4_O_3S:M17.6
TON    T103, 30
LRD
A      F_KQ4_C_10S:M17.7
TON    T104, 600
LPP
A      F_KQ4_C_5S:M18.0
TON    T105, 50
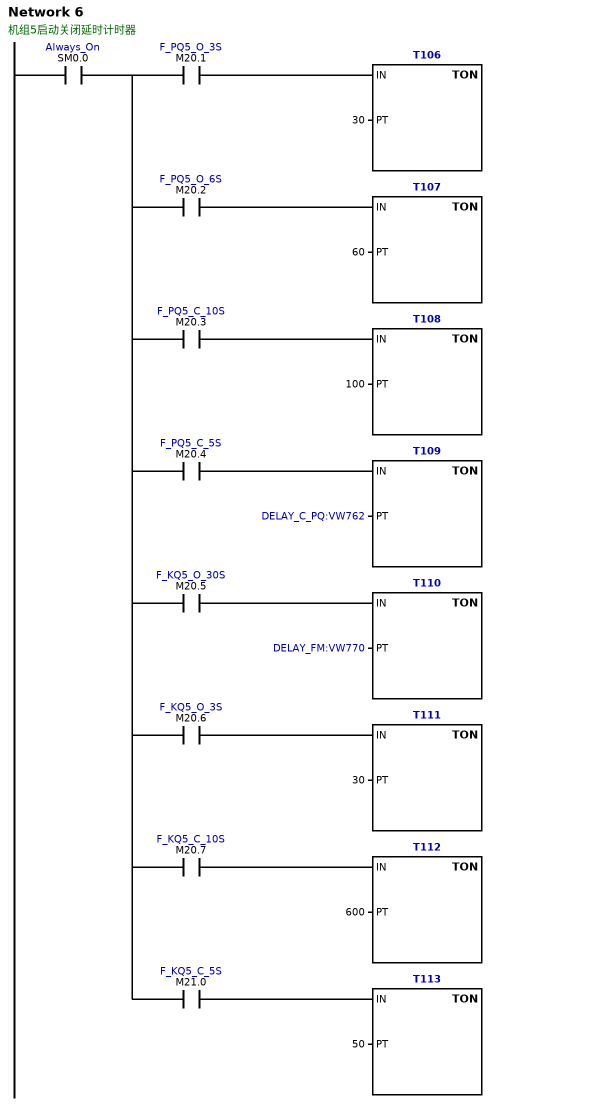
Network 6
// 机组5启动关闭延时计时器
LD     Always_On:SM0.0
LPS
A      F_PQ5_O_3S:M20.1
TON    T106, 30
LRD
A      F_PQ5_O_6S:M20.2
TON    T107, 60
LRD
A      F_PQ5_C_10S:M20.3
TON    T108, 100
LRD
A      F_PQ5_C_5S:M20.4
TON    T109, DELAY_C_PQ:VW762
LRD
A      F_KQ5_O_30S:M20.5
TON    T110, DELAY_FM:VW770
LRD
A      F_KQ5_O_3S:M20.6
TON    T111, 30
LRD
A      F_KQ5_C_10S:M20.7
TON    T112, 600
LPP
A      F_KQ5_C_5S:M21.0
TON    T113, 50
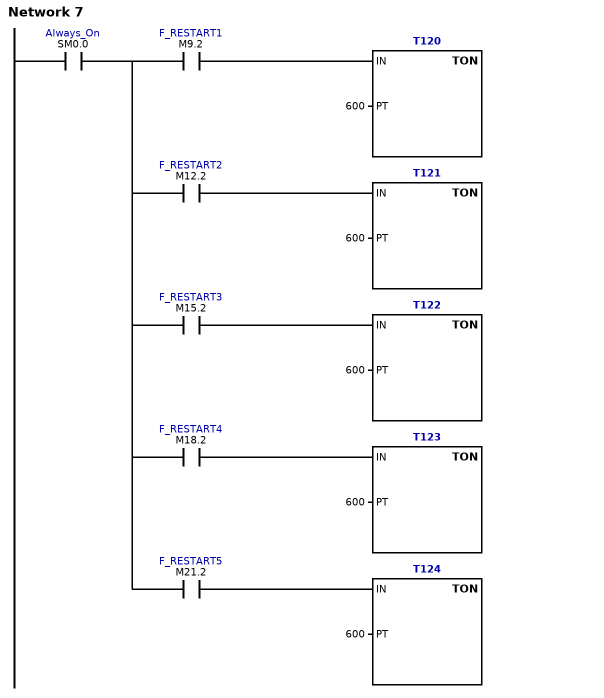
Network 7
LD     Always_On:SM0.0
LPS
A      F_RESTART1:M9.2
TON    T120, 600
LRD
A      F_RESTART2:M12.2
TON    T121, 600
LRD
A      F_RESTART3:M15.2
TON    T122, 600
LRD
A      F_RESTART4:M18.2
TON    T123, 600
LPP
A      F_RESTART5:M21.2
TON    T124, 600
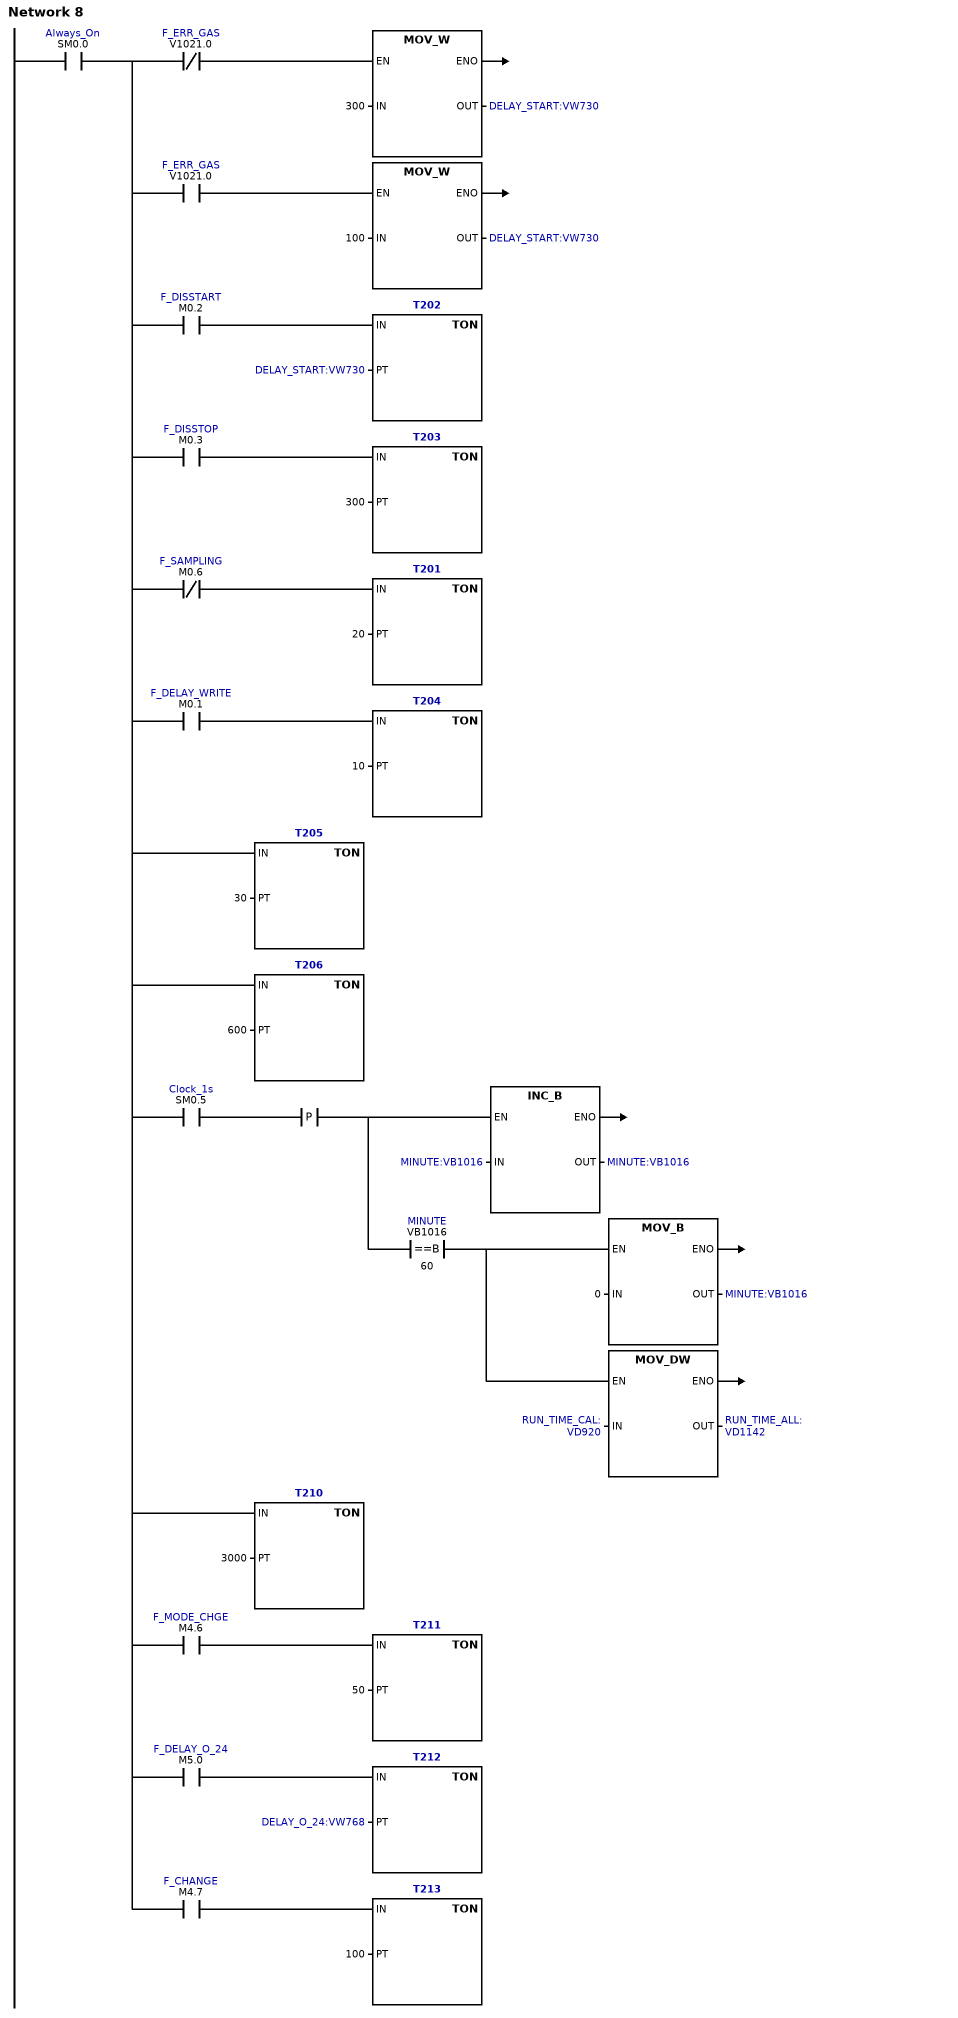
Network 8
LD     Always_On:SM0.0
LPS
AN     F_ERR_GAS:V1021.0
MOVW   300, DELAY_START:VW730
LRD
A      F_ERR_GAS:V1021.0
MOVW   100, DELAY_START:VW730
LRD
A      F_DISSTART:M0.2
TON    T202, DELAY_START:VW730
LRD
A      F_DISSTOP:M0.3
TON    T203, 300
LRD
AN     F_SAMPLING:M0.6
TON    T201, 20
LRD
A      F_DELAY_WRITE:M0.1
TON    T204, 10
LRD
TON    T205, 30
LRD
TON    T206, 600
LRD
A      Clock_1s:SM0.5
EU
INCB   MINUTE:VB1016
AB=    MINUTE:VB1016, 60
MOVB   0, MINUTE:VB1016
MOVD   RUN_TIME_CAL:VD920, RUN_TIME_ALL:VD1142
LPP
LPS
TON    T210, 3000
A      F_MODE_CHGE:M4.6
TON    T211, 50
LRD
A      F_DELAY_O_24:M5.0
TON    T212, DELAY_O_24:VW768
LPP
A      F_CHANGE:M4.7
TON    T213, 100
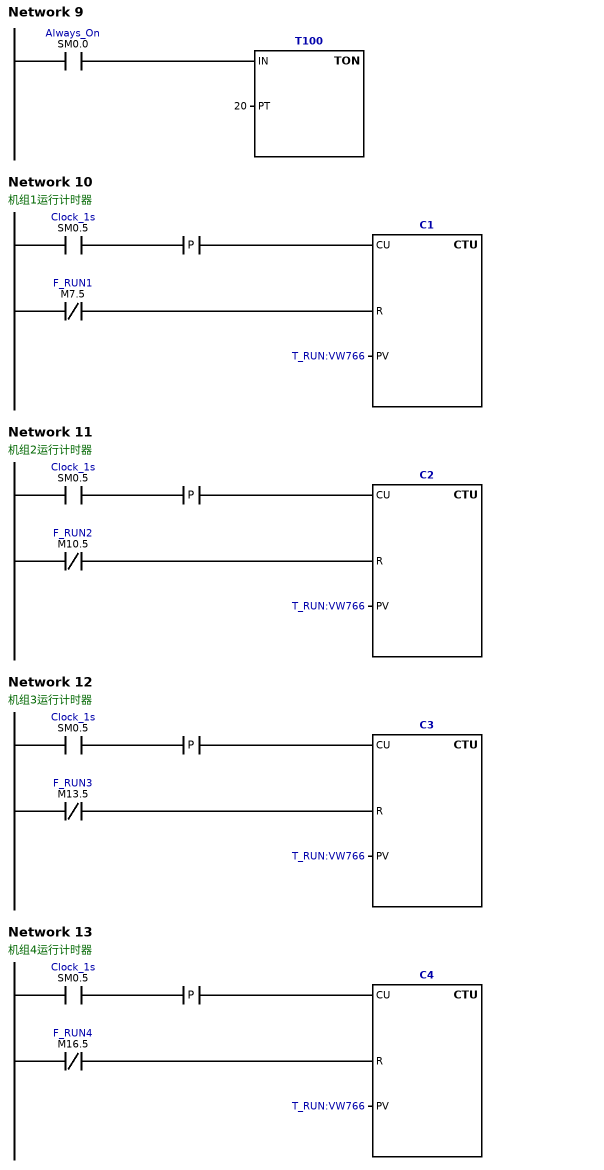
Network 9
LD     Always_On:SM0.0
TON    T100, 20
Network 10 //  
// 机组1运行计时器
LD     Clock_1s:SM0.5
EU
LDN    F_RUN1:M7.5
CTU    C1, T_RUN:VW766
Network 11 //  
// 机组2运行计时器
LD     Clock_1s:SM0.5
EU
LDN    F_RUN2:M10.5
CTU    C2, T_RUN:VW766
Network 12 //  
// 机组3运行计时器
LD     Clock_1s:SM0.5
EU
LDN    F_RUN3:M13.5
CTU    C3, T_RUN:VW766
Network 13 //  
// 机组4运行计时器
LD     Clock_1s:SM0.5
EU
LDN    F_RUN4:M16.5
CTU    C4, T_RUN:VW766
